FUNCTION_BLOCK CAerationLogic (* Composite Function Block Type *)
  (* Standard: 61499-2 *)
  (* Version 0.0, 10/24/2023, SESA685388, Schneider Electric, template *)
  PACKAGE SE.Nereda;
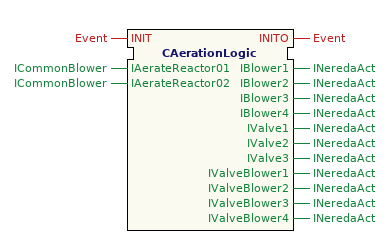
  EVENT_INPUT
    INIT; (* Initialization Request *)
  END_EVENT
  EVENT_OUTPUT
    INITO; (* Initialization Confirm *)
  END_EVENT
  SOCKETS
    IAerateReactor01 : ICommonBlower;
    IAerateReactor02 : ICommonBlower;
  END_SOCKETS
  PLUGS
    IBlower1 : INeredaAct;
    IBlower2 : INeredaAct;
    IBlower3 : INeredaAct;
    IBlower4 : INeredaAct;
    IValve1 : INeredaAct;
    IValve2 : INeredaAct;
    IValve3 : INeredaAct;
    IValveBlower1 : INeredaAct;
    IValveBlower2 : INeredaAct;
    IValveBlower3 : INeredaAct;
    IValveBlower4 : INeredaAct;
  END_PLUGS
  (* 01 - FUNCTIONNAL INPUT INTERFACE *)
  (* 00 - INITIALIZATION *)
  (* 05 - LOGIC *)
  (* 06 - HMI INTERFACE *)
  (* CommandLogic *)
  (* 02 - FUNCTIONNAL OUTPUT INTERFACE *)
  (* Capacity Sp *)
  FBS
    CommandLogicBL1BL4 : CAerationLogicBasic;
    Blower1Cmd_Smooth : boolValueChanged;
    Blower2Cmd_Smooth : boolValueChanged;
    IThis : CAerationLogic_HMI(QI := TRUE);
    Blower1Cmd : BOOL2INT;
    Blower2Cmd : BOOL2INT;
    Blower3Cmd_Smooth : boolValueChanged;
    Blower4Cmd_Smooth : boolValueChanged;
    Blower3Cmd : BOOL2INT;
    Blower4Cmd : BOOL2INT;
    Valve1Cmd_Smooth : boolValueChanged;
    Valve1Cmd : BOOL2INT;
    Valve2Cmd_Smooth : boolValueChanged;
    Valve3Cmd_Smooth : boolValueChanged;
    Valve2Cmd : BOOL2INT;
    Valve3Cmd : BOOL2INT;
    CommandLogicBL2BL3 : CAerationLogicBasic2;
    CapacitySp_Header1 : NeredaCapacitySpToCBlowersSp;
    CapacitySp_Header2 : NeredaCapacitySpToCBlowersSp;
    BL2AndBL3Manager : CAerationActCmd;
    EventSmooth : RetriggerEvent(pin_CFF51EFF0A91DC53 := 3, pin_FDD5DC24A8674AF6 := T#100ms);
    BlowerValve2Cmd_Smooth1 : boolValueChanged;
    BlowerValve4Cmd_Smooth1 : boolValueChanged;
    BlowerValve2Cmd1 : BOOL2INT;
    BlowerValve4Cmd1 : BOOL2INT;
    BlowerValve1Cmd_Smooth1 : boolValueChanged;
    BlowerValve3Cmd_Smooth1 : boolValueChanged;
    BlowerValve1Cmd1 : BOOL2INT;
    BlowerValve3Cmd1 : BOOL2INT;
    C2Time_H1 : E_DELAY;
    C3Time_H1 : E_DELAY;
    C2Time_H2 : E_DELAY;
    C3Time_H2 : E_DELAY;
  END_FBS
  EVENT_CONNECTIONS
    CommandLogicBL1BL4.B804F7AE49CF3E15 TO Blower1Cmd_Smooth.REQ;
    Blower1Cmd_Smooth.CHD TO Blower1Cmd.DD5870AA881150BB;
    Blower2Cmd_Smooth.CHD TO Blower2Cmd.DD5870AA881150BB;
    Blower3Cmd_Smooth.CHD TO Blower3Cmd.DD5870AA881150BB;
    Blower4Cmd_Smooth.CHD TO Blower4Cmd.DD5870AA881150BB;
    Valve1Cmd_Smooth.CHD TO Valve1Cmd.DD5870AA881150BB;
    Valve2Cmd_Smooth.CHD TO Valve2Cmd.DD5870AA881150BB;
    Valve3Cmd_Smooth.CHD TO Valve3Cmd.DD5870AA881150BB;
    Blower1Cmd_Smooth.CNF TO Blower2Cmd_Smooth.REQ;
    Blower2Cmd_Smooth.CNF TO Blower3Cmd_Smooth.REQ;
    Blower3Cmd_Smooth.CNF TO Blower4Cmd_Smooth.REQ;
    Blower4Cmd_Smooth.CNF TO Valve1Cmd_Smooth.REQ;
    Valve1Cmd_Smooth.CNF TO Valve2Cmd_Smooth.REQ;
    Valve2Cmd_Smooth.CNF TO Valve3Cmd_Smooth.REQ;
    Blower1Cmd.6FC99A5BD1C38561 TO IBlower1.0F1CDF9A9B4A227A;
    Blower2Cmd.6FC99A5BD1C38561 TO IBlower2.0F1CDF9A9B4A227A;
    Blower3Cmd.6FC99A5BD1C38561 TO IBlower3.0F1CDF9A9B4A227A;
    Blower4Cmd.6FC99A5BD1C38561 TO IBlower4.0F1CDF9A9B4A227A;
    Valve1Cmd.6FC99A5BD1C38561 TO IValve1.0F1CDF9A9B4A227A;
    Valve2Cmd.6FC99A5BD1C38561 TO IValve2.0F1CDF9A9B4A227A;
    Valve3Cmd.6FC99A5BD1C38561 TO IValve3.0F1CDF9A9B4A227A;
    IAerateReactor01.START_BLOWER TO CommandLogicBL1BL4.D2C11A8772DD75BE;
    IAerateReactor02.START_BLOWER TO CommandLogicBL1BL4.D2C11A8772DD75BE;
    IBlower1.9CD053F8408797ED TO IAerateReactor01.FB_BLOWER;
    IBlower1.CC753684FA882790 TO IAerateReactor01.FB_BLOWER_AVAILABLE;
    IBlower4.9CD053F8408797ED TO IAerateReactor02.FB_BLOWER;
    IBlower4.CC753684FA882790 TO IAerateReactor02.FB_BLOWER_AVAILABLE;
    IBlower1.9CD053F8408797ED TO CommandLogicBL1BL4.13BA3066C47C3D65;
    IBlower2.9CD053F8408797ED TO CommandLogicBL1BL4.13BA3066C47C3D65;
    IBlower3.9CD053F8408797ED TO CommandLogicBL1BL4.13BA3066C47C3D65;
    IBlower4.9CD053F8408797ED TO CommandLogicBL1BL4.13BA3066C47C3D65;
    IBlower1.CC753684FA882790 TO CommandLogicBL1BL4.C2CA1F9B44AEDC08;
    IBlower2.CC753684FA882790 TO CommandLogicBL1BL4.C2CA1F9B44AEDC08;
    IBlower3.CC753684FA882790 TO CommandLogicBL1BL4.C2CA1F9B44AEDC08;
    IBlower4.CC753684FA882790 TO CommandLogicBL1BL4.C2CA1F9B44AEDC08;
    IAerateReactor01.FLOW_SP_BLOWER TO CommandLogicBL1BL4.BF57157246C0E97B;
    IAerateReactor02.FLOW_SP_BLOWER TO CommandLogicBL1BL4.BF57157246C0E97B;
    IAerateReactor01.START_BLOWER TO CommandLogicBL2BL3.D2C11A8772DD75BE;
    IAerateReactor02.START_BLOWER TO CommandLogicBL2BL3.D2C11A8772DD75BE;
    IBlower1.CC753684FA882790 TO CommandLogicBL2BL3.D2C11A8772DD75BE;
    IBlower2.CC753684FA882790 TO CommandLogicBL2BL3.D2C11A8772DD75BE;
    IBlower3.CC753684FA882790 TO CommandLogicBL2BL3.D2C11A8772DD75BE;
    IBlower4.CC753684FA882790 TO CommandLogicBL2BL3.D2C11A8772DD75BE;
    IValve1.CC753684FA882790 TO CommandLogicBL2BL3.D2C11A8772DD75BE;
    IValve3.CC753684FA882790 TO CommandLogicBL2BL3.D2C11A8772DD75BE;
    IValve2.CC753684FA882790 TO CommandLogicBL2BL3.D2C11A8772DD75BE;
    IAerateReactor01.START_BLOWER TO CapacitySp_Header1.D0388ADF8D5604CA;
    IAerateReactor01.FLOW_SP_BLOWER TO CapacitySp_Header1.D0388ADF8D5604CA;
    IAerateReactor02.START_BLOWER TO CapacitySp_Header2.D0388ADF8D5604CA;
    IAerateReactor02.FLOW_SP_BLOWER TO CapacitySp_Header2.D0388ADF8D5604CA;
    CapacitySp_Header1.CNF TO IBlower1.1E00729184986247;
    CapacitySp_Header2.CNF TO IBlower4.1E00729184986247;
    BL2AndBL3Manager.71502B44797BB7D6 TO IBlower2.1E00729184986247;
    BL2AndBL3Manager.71502B44797BB7D6 TO IBlower3.1E00729184986247;
    CapacitySp_Header1.CNF TO CommandLogicBL2BL3.D2C11A8772DD75BE;
    CapacitySp_Header2.CNF TO CommandLogicBL2BL3.D2C11A8772DD75BE;
    CommandLogicBL2BL3.B804F7AE49CF3E15 TO EventSmooth.2BC1963D96179493;
    IBlower1.9CD053F8408797ED TO CommandLogicBL2BL3.D2C11A8772DD75BE;
    IBlower2.9CD053F8408797ED TO CommandLogicBL2BL3.D2C11A8772DD75BE;
    IBlower3.9CD053F8408797ED TO CommandLogicBL2BL3.D2C11A8772DD75BE;
    IBlower4.9CD053F8408797ED TO CommandLogicBL2BL3.D2C11A8772DD75BE;
    IValve1.9CD053F8408797ED TO CommandLogicBL2BL3.D2C11A8772DD75BE;
    IValve3.9CD053F8408797ED TO CommandLogicBL2BL3.D2C11A8772DD75BE;
    IValve2.9CD053F8408797ED TO CommandLogicBL2BL3.D2C11A8772DD75BE;
    EventSmooth.4002AEF0814D09CF TO BL2AndBL3Manager.D2C11A8772DD75BE;
    BlowerValve2Cmd_Smooth1.CHD TO BlowerValve2Cmd1.DD5870AA881150BB;
    BlowerValve4Cmd_Smooth1.CHD TO BlowerValve4Cmd1.DD5870AA881150BB;
    BlowerValve1Cmd_Smooth1.CHD TO BlowerValve1Cmd1.DD5870AA881150BB;
    BlowerValve3Cmd_Smooth1.CHD TO BlowerValve3Cmd1.DD5870AA881150BB;
    BlowerValve2Cmd_Smooth1.CNF TO BlowerValve4Cmd_Smooth1.REQ;
    BlowerValve4Cmd_Smooth1.CNF TO BlowerValve1Cmd_Smooth1.REQ;
    BlowerValve1Cmd_Smooth1.CNF TO BlowerValve3Cmd_Smooth1.REQ;
    BL2AndBL3Manager.B804F7AE49CF3E15 TO BlowerValve2Cmd_Smooth1.REQ;
    CommandLogicBL1BL4.B804F7AE49CF3E15 TO BlowerValve4Cmd_Smooth1.REQ;
    CommandLogicBL1BL4.B804F7AE49CF3E15 TO BlowerValve1Cmd_Smooth1.REQ;
    BlowerValve4Cmd1.6FC99A5BD1C38561 TO IValveBlower4.0F1CDF9A9B4A227A;
    BlowerValve2Cmd1.6FC99A5BD1C38561 TO IValveBlower2.0F1CDF9A9B4A227A;
    BlowerValve3Cmd1.6FC99A5BD1C38561 TO IValveBlower3.0F1CDF9A9B4A227A;
    BlowerValve1Cmd1.6FC99A5BD1C38561 TO IValveBlower1.0F1CDF9A9B4A227A;
    IValveBlower1.CC753684FA882790 TO CommandLogicBL1BL4.77D7986251D66128;
    IValveBlower1.9CD053F8408797ED TO CommandLogicBL1BL4.E57CC257F577A1D0;
    IValveBlower4.9CD053F8408797ED TO CommandLogicBL1BL4.E57CC257F577A1D0;
    IValveBlower4.CC753684FA882790 TO CommandLogicBL1BL4.77D7986251D66128;
    IValveBlower2.9CD053F8408797ED TO BL2AndBL3Manager.D2C11A8772DD75BE;
    IValveBlower3.9CD053F8408797ED TO BL2AndBL3Manager.D2C11A8772DD75BE;
    IValveBlower2.CC753684FA882790 TO BL2AndBL3Manager.D2C11A8772DD75BE;
    INIT TO IThis.73B62E902A5807A1;
    IThis.F68012C9A80C276B TO IThis.559778F4ADF98A31;
    IThis.F68012C9A80C276B TO INITO;
    IThis.3F1A2A449466611E TO CommandLogicBL2BL3.D2C11A8772DD75BE;
    IThis.3F1A2A449466611E TO CapacitySp_Header1.D0388ADF8D5604CA;
    IThis.3F1A2A449466611E TO CapacitySp_Header2.D0388ADF8D5604CA;
    CapacitySp_Header1.C8BBF715CC922495 TO C2Time_H1.START;
    CapacitySp_Header2.C8BBF715CC922495 TO C2Time_H2.START;
    CapacitySp_Header1.C529EC06887E5F22 TO C3Time_H1.START;
    CapacitySp_Header2.C529EC06887E5F22 TO C3Time_H2.START;
    C2Time_H1.EO TO CapacitySp_Header1.C290CA59E2E76CE7;
    C3Time_H1.EO TO CapacitySp_Header1.928BD6855BDB8CD4;
    C2Time_H2.EO TO CapacitySp_Header2.C290CA59E2E76CE7;
    C3Time_H2.EO TO CapacitySp_Header2.928BD6855BDB8CD4;
    CapacitySp_Header1.CNF TO BL2AndBL3Manager.D2C11A8772DD75BE;
    CapacitySp_Header2.CNF TO BL2AndBL3Manager.D2C11A8772DD75BE;
    CommandLogicBL2BL3.B804F7AE49CF3E15 TO CapacitySp_Header2.D0388ADF8D5604CA;
    CommandLogicBL2BL3.B804F7AE49CF3E15 TO CapacitySp_Header1.D0388ADF8D5604CA;
    IBlower2.9CD053F8408797ED TO BL2AndBL3Manager.D2C11A8772DD75BE;
    IBlower3.9CD053F8408797ED TO BL2AndBL3Manager.D2C11A8772DD75BE;
    IValve1.9CD053F8408797ED TO BL2AndBL3Manager.D2C11A8772DD75BE;
    IValve1.CC753684FA882790 TO BL2AndBL3Manager.D2C11A8772DD75BE;
    IValveBlower1.CC753684FA882790 TO BL2AndBL3Manager.D2C11A8772DD75BE;
    IValveBlower1.9CD053F8408797ED TO BL2AndBL3Manager.D2C11A8772DD75BE;
    IBlower1.9CD053F8408797ED TO BL2AndBL3Manager.D2C11A8772DD75BE;
    IBlower1.CC753684FA882790 TO BL2AndBL3Manager.D2C11A8772DD75BE;
    IBlower2.CC753684FA882790 TO BL2AndBL3Manager.D2C11A8772DD75BE;
    IValve2.9CD053F8408797ED TO BL2AndBL3Manager.D2C11A8772DD75BE;
    IValve2.CC753684FA882790 TO BL2AndBL3Manager.D2C11A8772DD75BE;
    IValve3.CC753684FA882790 TO BL2AndBL3Manager.D2C11A8772DD75BE;
    IValve3.9CD053F8408797ED TO BL2AndBL3Manager.D2C11A8772DD75BE;
    IBlower3.CC753684FA882790 TO BL2AndBL3Manager.D2C11A8772DD75BE;
    IBlower4.9CD053F8408797ED TO BL2AndBL3Manager.D2C11A8772DD75BE;
    IBlower4.CC753684FA882790 TO BL2AndBL3Manager.D2C11A8772DD75BE;
    IValveBlower4.9CD053F8408797ED TO BL2AndBL3Manager.D2C11A8772DD75BE;
    IValveBlower4.CC753684FA882790 TO BL2AndBL3Manager.D2C11A8772DD75BE;
    IValveBlower3.CC753684FA882790 TO BL2AndBL3Manager.D2C11A8772DD75BE;
    IValveBlower3.9CD053F8408797ED TO CommandLogicBL2BL3.D2C11A8772DD75BE;
    IValveBlower3.CC753684FA882790 TO CommandLogicBL2BL3.D2C11A8772DD75BE;
    IValveBlower2.9CD053F8408797ED TO CommandLogicBL2BL3.D2C11A8772DD75BE;
    IValveBlower2.CC753684FA882790 TO CommandLogicBL2BL3.D2C11A8772DD75BE;
    IValveBlower1.CC753684FA882790 TO CommandLogicBL2BL3.D2C11A8772DD75BE;
    IValveBlower1.9CD053F8408797ED TO CommandLogicBL2BL3.D2C11A8772DD75BE;
    IValveBlower4.9CD053F8408797ED TO CommandLogicBL2BL3.D2C11A8772DD75BE;
    IValveBlower4.CC753684FA882790 TO CommandLogicBL2BL3.D2C11A8772DD75BE;
    CommandLogicBL2BL3.B804F7AE49CF3E15 TO BL2AndBL3Manager.D2C11A8772DD75BE;
    BL2AndBL3Manager.B804F7AE49CF3E15 TO Valve1Cmd_Smooth.REQ;
    BL2AndBL3Manager.B804F7AE49CF3E15 TO Valve2Cmd_Smooth.REQ;
    BL2AndBL3Manager.B804F7AE49CF3E15 TO Valve3Cmd_Smooth.REQ;
    BL2AndBL3Manager.B804F7AE49CF3E15 TO Blower2Cmd_Smooth.REQ;
    BL2AndBL3Manager.B804F7AE49CF3E15 TO BlowerValve3Cmd_Smooth1.REQ;
    BL2AndBL3Manager.B804F7AE49CF3E15 TO Blower3Cmd_Smooth.REQ;
  END_CONNECTIONS
  DATA_CONNECTIONS
    CommandLogicBL1BL4.6F30DD159F832B4D TO Blower1Cmd_Smooth.Input;
    Blower1Cmd_Smooth.Output TO Blower1Cmd.4573FC8F228EB71D;
    Blower2Cmd_Smooth.Output TO Blower2Cmd.4573FC8F228EB71D;
    IBlower1.D83B5BDEFA4D797C TO IAerateReactor01.FBStop;
    IBlower1.B762734C094A7162 TO IAerateReactor01.FBStart;
    IBlower4.D83B5BDEFA4D797C TO IAerateReactor02.FBStop;
    IBlower4.B762734C094A7162 TO IAerateReactor02.FBStart;
    Blower3Cmd_Smooth.Output TO Blower3Cmd.4573FC8F228EB71D;
    Blower4Cmd_Smooth.Output TO Blower4Cmd.4573FC8F228EB71D;
    Valve1Cmd_Smooth.Output TO Valve1Cmd.4573FC8F228EB71D;
    Valve2Cmd_Smooth.Output TO Valve2Cmd.4573FC8F228EB71D;
    Valve3Cmd_Smooth.Output TO Valve3Cmd.4573FC8F228EB71D;
    CommandLogicBL1BL4.888716159CBC3FDC TO Blower4Cmd_Smooth.Input;
    Blower1Cmd.A6DEF5F9C27C1848 TO IBlower1.710D7FC54EE3F35A;
    Blower2Cmd.A6DEF5F9C27C1848 TO IBlower2.710D7FC54EE3F35A;
    Blower3Cmd.A6DEF5F9C27C1848 TO IBlower3.710D7FC54EE3F35A;
    Blower4Cmd.A6DEF5F9C27C1848 TO IBlower4.710D7FC54EE3F35A;
    Valve1Cmd.A6DEF5F9C27C1848 TO IValve1.710D7FC54EE3F35A;
    Valve2Cmd.A6DEF5F9C27C1848 TO IValve2.710D7FC54EE3F35A;
    Valve3Cmd.A6DEF5F9C27C1848 TO IValve3.710D7FC54EE3F35A;
    IAerateReactor01.StartBlower TO CommandLogicBL1BL4.B2CC9DAB470B3A98;
    IAerateReactor02.StartBlower TO CommandLogicBL1BL4.1AEE3F619E7084DB;
    IBlower1.8A8A07EFCDA1443C TO IAerateReactor01.FBBlowersAbailable;
    IBlower4.8A8A07EFCDA1443C TO IAerateReactor02.FBBlowersAbailable;
    IBlower1.D83B5BDEFA4D797C TO CommandLogicBL1BL4.CF3BA6B848432326;
    IBlower4.D83B5BDEFA4D797C TO CommandLogicBL1BL4.7970F58D086A71AC;
    IBlower1.B762734C094A7162 TO CommandLogicBL1BL4.AF84CB02D2B46EA7;
    IBlower4.B762734C094A7162 TO CommandLogicBL1BL4.A0D7CFCA437A0AE1;
    IBlower1.8A8A07EFCDA1443C TO CommandLogicBL1BL4.0D2984DD8432BDE4;
    IBlower4.8A8A07EFCDA1443C TO CommandLogicBL1BL4.71560028BEB1A1C1;
    IAerateReactor01.FlowSPBlower TO CommandLogicBL1BL4.09FC2180130EA7A8;
    IAerateReactor02.FlowSPBlower TO CommandLogicBL1BL4.4A7C96523834A9A5;
    BL2AndBL3Manager.50D97D2FBAA8D1BB TO Blower2Cmd_Smooth.Input;
    BL2AndBL3Manager.101F312D51A39512 TO Blower3Cmd_Smooth.Input;
    BL2AndBL3Manager.7162276D9F2FFFC0 TO Valve1Cmd_Smooth.Input;
    BL2AndBL3Manager.ED0ED021ACC74439 TO Valve2Cmd_Smooth.Input;
    BL2AndBL3Manager.17AB3608D374DB0E TO Valve3Cmd_Smooth.Input;
    IValve1.7F6CC7FEB9223DF3 TO BL2AndBL3Manager.3BA4286809D56F12;
    IValve1.A8D6C4A1FDCCA991 TO BL2AndBL3Manager.2F5A12506C1E3BF8;
    IValve2.7F6CC7FEB9223DF3 TO BL2AndBL3Manager.730E3F472BEC096F;
    IValve2.A8D6C4A1FDCCA991 TO BL2AndBL3Manager.4E9CCE0C08151AB9;
    IValve3.7F6CC7FEB9223DF3 TO BL2AndBL3Manager.877975637185E5E2;
    IValve3.A8D6C4A1FDCCA991 TO BL2AndBL3Manager.CF96F74CBA9BB4AF;
    IBlower2.8A8A07EFCDA1443C TO CommandLogicBL2BL3.266E7B658D2D8018;
    IBlower3.8A8A07EFCDA1443C TO CommandLogicBL2BL3.7D28FD8AC101CEE8;
    IAerateReactor01.StartBlower TO CommandLogicBL2BL3.B2CC9DAB470B3A98;
    IAerateReactor02.StartBlower TO CommandLogicBL2BL3.1AEE3F619E7084DB;
    IAerateReactor01.FlowSPBlower TO CommandLogicBL2BL3.09FC2180130EA7A8;
    IAerateReactor02.FlowSPBlower TO CommandLogicBL2BL3.4A7C96523834A9A5;
    IAerateReactor01.FlowSPBlower TO CapacitySp_Header1.Setpoint;
    IAerateReactor02.FlowSPBlower TO CapacitySp_Header2.Setpoint;
    CapacitySp_Header1.SpeedBlower TO IBlower1.1BC103921BBFDA0B;
    CapacitySp_Header2.SpeedBlower TO IBlower4.1BC103921BBFDA0B;
    CapacitySp_Header1.SpeedBlower TO BL2AndBL3Manager.58EEDBE222456145;
    CapacitySp_Header2.SpeedBlower TO BL2AndBL3Manager.7ADECE91806B407A;
    BL2AndBL3Manager.8CE2038B5C8422BA TO IBlower2.1BC103921BBFDA0B;
    BL2AndBL3Manager.C40FC192AC89DE17 TO IBlower3.1BC103921BBFDA0B;
    IBlower1.8A8A07EFCDA1443C TO CommandLogicBL2BL3.F39CADEC2A13420A;
    IBlower4.8A8A07EFCDA1443C TO CommandLogicBL2BL3.BD31FDCAB4D0C603;
    CommandLogicBL2BL3.4F511D89CFAD767B TO BL2AndBL3Manager.4DF2BEC52A74E46B;
    CommandLogicBL2BL3.FE3CA976DB528EC5 TO BL2AndBL3Manager.DBE2A8D701392E9A;
    CommandLogicBL2BL3.C27B618F80BE71A0 TO BL2AndBL3Manager.A67F51A8CEE7381C;
    CommandLogicBL2BL3.DFDB6D6DAFE2FA40 TO BL2AndBL3Manager.748CEDEC849105C0;
    IBlower2.B762734C094A7162 TO BL2AndBL3Manager.09DD17EC8B73785F;
    IBlower2.D83B5BDEFA4D797C TO BL2AndBL3Manager.01BBAA5934ACED59;
    IBlower3.B762734C094A7162 TO BL2AndBL3Manager.15986335CE8A5236;
    IBlower3.D83B5BDEFA4D797C TO BL2AndBL3Manager.C7753AC130D578A9;
    IValve1.8A8A07EFCDA1443C TO BL2AndBL3Manager.FF754D33E60B1E14;
    IValve2.8A8A07EFCDA1443C TO BL2AndBL3Manager.041D8CCDD94E4A77;
    IValve3.8A8A07EFCDA1443C TO BL2AndBL3Manager.D8974B00E26B10C6;
    IAerateReactor01.StartBlower TO BL2AndBL3Manager.9A96836ABFCFF66A;
    IAerateReactor02.StartBlower TO BL2AndBL3Manager.6B729D4387003A21;
    BlowerValve2Cmd_Smooth1.Output TO BlowerValve2Cmd1.4573FC8F228EB71D;
    BlowerValve4Cmd_Smooth1.Output TO BlowerValve4Cmd1.4573FC8F228EB71D;
    BlowerValve1Cmd_Smooth1.Output TO BlowerValve1Cmd1.4573FC8F228EB71D;
    BlowerValve3Cmd_Smooth1.Output TO BlowerValve3Cmd1.4573FC8F228EB71D;
    BlowerValve1Cmd1.A6DEF5F9C27C1848 TO IValveBlower1.710D7FC54EE3F35A;
    BlowerValve2Cmd1.A6DEF5F9C27C1848 TO IValveBlower2.710D7FC54EE3F35A;
    BlowerValve3Cmd1.A6DEF5F9C27C1848 TO IValveBlower3.710D7FC54EE3F35A;
    BlowerValve4Cmd1.A6DEF5F9C27C1848 TO IValveBlower4.710D7FC54EE3F35A;
    IValveBlower1.7F6CC7FEB9223DF3 TO CommandLogicBL1BL4.DD539EBA296107FA;
    IValveBlower1.A8D6C4A1FDCCA991 TO CommandLogicBL1BL4.602F392F126AA85C;
    IValveBlower1.8A8A07EFCDA1443C TO CommandLogicBL1BL4.C6EDB0A1C3E2CD9E;
    IValveBlower4.7F6CC7FEB9223DF3 TO CommandLogicBL1BL4.75EDF7C081990EBA;
    IValveBlower4.A8D6C4A1FDCCA991 TO CommandLogicBL1BL4.D59A94C6C1D30D86;
    IValveBlower4.8A8A07EFCDA1443C TO CommandLogicBL1BL4.36717EB085C1DD5C;
    CommandLogicBL1BL4.6A904F40D20029A1 TO BlowerValve1Cmd_Smooth1.Input;
    CommandLogicBL1BL4.064AFCAEB0DD5723 TO BlowerValve4Cmd_Smooth1.Input;
    IValveBlower2.7F6CC7FEB9223DF3 TO BL2AndBL3Manager.54110732FC12EAAC;
    IValveBlower2.A8D6C4A1FDCCA991 TO BL2AndBL3Manager.8610CAD1FF35313D;
    IValveBlower3.7F6CC7FEB9223DF3 TO BL2AndBL3Manager.446B908A6A6E947E;
    IValveBlower3.A8D6C4A1FDCCA991 TO BL2AndBL3Manager.B5780401553C42A4;
    IValveBlower2.8A8A07EFCDA1443C TO BL2AndBL3Manager.5A95514FC9A40F7D;
    IValveBlower3.8A8A07EFCDA1443C TO BL2AndBL3Manager.03F395656869D664;
    BL2AndBL3Manager.56C8D5F7E1B68F58 TO BlowerValve2Cmd_Smooth1.Input;
    BL2AndBL3Manager.D78C80681718ACEF TO BlowerValve3Cmd_Smooth1.Input;
    IThis.1A24AFB83170123C TO CommandLogicBL2BL3.BB0AA5D7C20FC6DC;
    IThis.1A24AFB83170123C TO CapacitySp_Header1.366DF9C08522C788;
    IThis.1A24AFB83170123C TO CapacitySp_Header2.366DF9C08522C788;
    IThis.35C7139260F4D47E TO C2Time_H1.DT;
    IThis.606E767CD2B530F5 TO CapacitySp_Header1.0E6B92BFBD466C31;
    IThis.606E767CD2B530F5 TO CapacitySp_Header2.0E6B92BFBD466C31;
    IThis.A8DDE26075A11F35 TO CommandLogicBL2BL3.82E6F957CA34CE22;
    IThis.A8DDE26075A11F35 TO CapacitySp_Header1.9458FDB1B841EBF6;
    IThis.A8DDE26075A11F35 TO CapacitySp_Header2.9458FDB1B841EBF6;
    IThis.ADACDD2051362C28 TO C3Time_H2.DT;
    IThis.35C7139260F4D47E TO C2Time_H2.DT;
    IThis.ADACDD2051362C28 TO C3Time_H1.DT;
    IThis.606E767CD2B530F5 TO CommandLogicBL2BL3.15021417A9DDC3CD;
    CommandLogicBL2BL3.1B895462E4166559 TO CapacitySp_Header1.1FE73434323A3C55;
    CommandLogicBL2BL3.F7BB9EFC676442B0 TO CapacitySp_Header2.1FE73434323A3C55;
    CommandLogicBL2BL3.CF61785EEFC670F6 TO CapacitySp_Header2.F347E80EA65C1CE5;
    CommandLogicBL2BL3.666629205E956536 TO CapacitySp_Header1.F347E80EA65C1CE5;
    IBlower1.B762734C094A7162 TO CommandLogicBL2BL3.CB32EC934DF76E18;
    IBlower2.B762734C094A7162 TO CommandLogicBL2BL3.8557D5BDB3557853;
    IBlower3.B762734C094A7162 TO CommandLogicBL2BL3.987796B5153B8A12;
    IBlower4.B762734C094A7162 TO CommandLogicBL2BL3.6E6C99EFCC1CAE58;
    IValve1.7F6CC7FEB9223DF3 TO CommandLogicBL2BL3.ABE62E0DB94B9D1A;
    IValve1.8A8A07EFCDA1443C TO CommandLogicBL2BL3.E25FE5C20B781EFF;
    IValve2.7F6CC7FEB9223DF3 TO CommandLogicBL2BL3.7E8E090D1C9E6C5A;
    IValve2.8A8A07EFCDA1443C TO CommandLogicBL2BL3.A452A22B1B0D495A;
    IValve3.7F6CC7FEB9223DF3 TO CommandLogicBL2BL3.C25A6B8F9DCB96E0;
    IValve3.8A8A07EFCDA1443C TO CommandLogicBL2BL3.DF20542FEA597588;
    IValveBlower2.7F6CC7FEB9223DF3 TO CommandLogicBL2BL3.1030013A11257D60;
    IValveBlower2.8A8A07EFCDA1443C TO CommandLogicBL2BL3.EB34E2DAA4465570;
    IValveBlower3.7F6CC7FEB9223DF3 TO CommandLogicBL2BL3.55B3DAAF979CC2E7;
    IValveBlower3.8A8A07EFCDA1443C TO CommandLogicBL2BL3.7FE01B1E5554C313;
    IValveBlower1.7F6CC7FEB9223DF3 TO CommandLogicBL2BL3.99B4843F7ED498C4;
    IValveBlower1.8A8A07EFCDA1443C TO CommandLogicBL2BL3.68E67740CA57E71D;
    IValveBlower4.7F6CC7FEB9223DF3 TO CommandLogicBL2BL3.3B81A0671CD7BCF6;
    IValveBlower4.8A8A07EFCDA1443C TO CommandLogicBL2BL3.C4B9BEEAC199E058;
  END_CONNECTIONS
END_FUNCTION_BLOCK
